{attribute addProperty BoxType "KL6224"}
{attribute addProperty Id "Channel_1Channel_BDA872B600"}
{attribute addProperty CRC "3598952469"}
{attribute addProperty SizeInBites "0"}
{attribute addProperty SizeInBytes "0"}
TYPE KL6224_D683A815 :
STRUCT
	{attribute addProperty Name "Channel_1"}
	Channel_1 : Channel_BDA872B6;
END_STRUCT
END_TYPE

(* stored: Version 1.2.0.0, ProductVersion 3.1.4024.9
   DUT KL6224_D683A815: Id {0c640133-4f85-498d-8616-05d64a563ff6} *)
